// TwinCAT 3 PLC project fliker
// libraries:
//   Tc2_Standard, * (Beckhoff Automation GmbH)
//   Tc2_System, * (Beckhoff Automation GmbH)
//   Tc2_Utilities, * (Beckhoff Automation GmbH)
//   Tc3_Module, * (Beckhoff Automation GmbH)
// project tree:
//   Global Variables/ Global_Variables.TcGVL, TwinCAT_Configuration.TcGVL, Variable_Configuration.TcGVL
//   / GlobalImagePool.TcGIPO (not stored)
//   POUs/ MAIN.TcPOU
//   Visualizations/ test.TcVIS

// ---- Global Variables/Global_Variables.TcGVL
{attribute 'Tc2GvlVarNames'}
VAR_GLOBAL
END_VAR

// ---- Global Variables/TwinCAT_Configuration.TcGVL
{attribute 'Tc2GvlVarNames'}
(* Generated automatically by TwinCAT - (read only) *)
VAR_CONFIG
	MAIN.push AT %IX0.0 : BOOL;	(*  ~ {LinkedWith:TIID^Device 2 (EtherCAT (v2.10 only))^Term 1 (EK1100)^Term 2 (EL1008)^Channel 2^Input} *)
END_VAR

// ---- Global Variables/Variable_Configuration.TcGVL
{attribute 'Tc2GvlVarNames'}
VAR_CONFIG
END_VAR

// ---- POUs/MAIN.TcPOU
PROGRAM MAIN
VAR
	tofftime : TON;
	tontime: TOF;
	Q: BOOL;
	Q2: BOOL;
	push AT %I* : BOOL;
	arrWaarde : ARRAY[1..2,1..10] OF STRING;
	fbTime : FB_LocalSystemTime := ( bEnable := TRUE, dwCycle := 1 );
	trigger: F_TRIG;
	X: INT;
END_VAR

fbTime();
trigger(CLK:= push);
tofftime(IN:= NOT Q, PT:= t#1s, Q=> Q2, ET=> );
tontime(IN:= Q2 , PT:= t#5s, Q=> Q, ET=> );

IF trigger.Q THEN
	FOR X :=10 TO 1 BY -1 DO
		arrWaarde[1,X] := arrWaarde[1,X-1];
		arrWaarde[2,X] := arrWaarde[2,X-1];
	END_FOR;
	arrWaarde[1,1] := SYSTEMTIME_TO_STRING(fbTime.systemTime);
	arrWaarde[2,1] := BOOL_TO_STRING(Q) ;
END_IF

END_PROGRAM

// ---- Visualizations/test.TcVIS
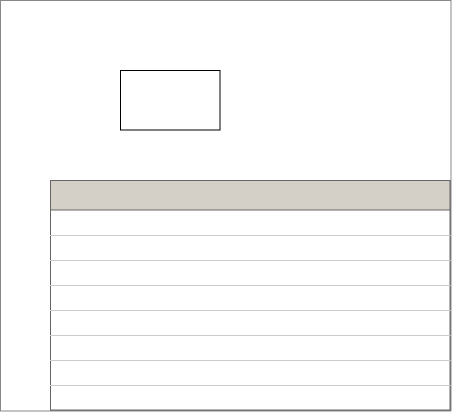
VISUALIZATION test  // 452x412
    Rectangle (120,70 100x60), colour toggle: MAIN.Q
    Table (50,180 400x230), data array: MAIN.arrWaarde
        p2232123230: MAIN.arrWaarde[1, INDEX]
        p511219082: MAIN.arrWaarde[2, INDEX]
END_VISUALIZATION
